{attribute 'linkalways'} 
{attribute 'no_explicit_call' := 'This FB is a CLASS and must be accessed using methods or properties'}
{attribute 'enable_dynamic_creation'}
FUNCTION_BLOCK _BOOL EXTENDS DatatypeBase
VAR
	localData : BOOL;
	activeData : REFERENCE TO BOOL REF= localData;
END_VAR

PROPERTY PUBLIC Address : PVOID
GET
Address := ADR(activeData);
END_GET
END_PROPERTY

METHOD PUBLIC ClearReference
VAR_INPUT
END_VAR
activeData REF= localData;
END_METHOD

METHOD PUBLIC Clone : I_Datatype
VAR
    pClone : POINTER TO _BOOL;
END_VAR
pClone := __NEW(_BOOL(InitialValue := Value));
Clone := pClone^;
END_METHOD

METHOD FB_init : BOOL
VAR_INPUT
	bInitRetains : BOOL; // if TRUE, the retain variables are initialized (warm start / cold start)
	bInCopyCode : BOOL;  // if TRUE, the instance afterwards gets moved into the copy code (online change)
	InitialValue : BOOL;
END_VAR
localData := InitialValue;
END_METHOD

METHOD PUBLIC MakeReferenceTo
VAR_INPUT
	ReferenceTarget : REFERENCE TO BOOL;
END_VAR
activeData REF= ReferenceTarget;
END_METHOD

METHOD PUBLIC SerializeWith
VAR_INPUT
	Serializer : I_Serializer;
END_VAR
Serializer.AddBool(activeData);
END_METHOD

PROPERTY PUBLIC Size : UDINT
GET
Size := SIZEOF(activeData);
END_GET
END_PROPERTY

METHOD TryDeserializeFrom : BOOL
VAR_INPUT
	Deserializer : I_Deserializer;
	Feedback : I_DeserializerFeedback;
END_VAR
TryDeserializeFrom := Deserializer.TryGetBool(activeData, Feedback);
END_METHOD

METHOD TryMakeReferenceTo : BOOL
VAR_INPUT
	Target : I_Datatype;
END_VAR
VAR
	pTargetData : POINTER TO BOOL;
END_VAR
IF NOT (Target.TypeName = TypeName) THEN
	RETURN;
END_IF

pTargetData := Target.Address;
activeData REF= pTargetData^;
TryMakeReferenceTo := TRUE;
END_METHOD

PROPERTY PUBLIC TypeName : T_MAXSTRING
GET
TypeName := 'BOOL';
END_GET
END_PROPERTY

PROPERTY PUBLIC Value : BOOL
GET
Value := activeData;
END_GET
SET
activeData := Value;
END_SET
END_PROPERTY

END_FUNCTION_BLOCK

(* stored: Version 1.1.0.1, ProductVersion 3.1.4024.12
   POU _BOOL: Id {32ecd87b-dc59-0e12-24dd-b9567367eb45}, SpecialFunc None
   Folder Constructor: Id {9a5835ce-e84d-08a5-0d36-04d775984943}
   Property Address: Id {a14dd81c-ebb8-0f68-0fcc-eabf0205b0fb}
   Get Get: Id {e18f823c-05db-0beb-1922-03bf1fa24519}
   Method ClearReference: Id {96b375be-40c5-03e2-1c98-9461aee7b003}
   Method Clone: Id {1b8d6504-b712-0ab3-0bf2-7a1fc0883766}
   Method FB_init: Id {51b5c943-33c7-0b59-1095-2fbe6237611e}
   Method MakeReferenceTo: Id {e61b5a40-d283-05bf-3d3d-ad5d5ebda2cb}
   Method SerializeWith: Id {f104fc17-3c44-0923-0d99-8a6eb4827d17}
   Property Size: Id {b786495b-9c2f-0ebd-3002-9d96d4ad3ce9}
   Get Get: Id {6b14d758-58f0-06a1-0a3f-696fd7a29696}
   Method TryDeserializeFrom: Id {433325ee-0af5-03f1-3a60-677bbbceb824}
   Method TryMakeReferenceTo: Id {22692f42-ea75-064b-2b93-009a42ef0e96}
   Property TypeName: Id {0105f59f-1385-094c-2744-f1892f3c172e}
   Get Get: Id {1981143b-b4f2-011d-378c-f413a2b65878}
   Property Value: Id {76b17b1c-172e-05c1-1aea-ad9e4a83b19d}
   Get Get: Id {146c5ec8-3aa7-0047-2d80-3317386dc124}
   Set Set: Id {e242f494-691c-0c1f-3d98-1ac3e3f69d6e} *)
